FUNCTION_BLOCK T_PMLSubUnitInfoCollection EXTENDS T_NamedBase IMPLEMENTS I_PMLSubUnitInfo
VAR
	_info : ST_PMLSubUnitInfo;
	baseCollection : T_CollectionBase;
END_VAR

METHOD AddUnit : BOOL
VAR_INPUT
	newUnit : I_PMLSubUnitInfo;
END_VAR
IF newUnit = 0 THEN
	LogError( 'Cannot AddUnit invalid ref' );
	RETURN;
END_IF

AddUnit := baseCollection.AddItem( newItem := CastToBase(newUnit) );
END_METHOD

METHOD PRIVATE CastToBase : I_InterfaceBase
VAR_INPUT
	Unit : I_PMLSubUnitInfo;
END_VAR
__QUERYINTERFACE(Unit, CastToBase);
END_METHOD

METHOD CastToType : I_PMLSubUnitInfo
VAR_INPUT
	Base : I_InterfaceBase;
END_VAR
__QUERYINTERFACE(Base, CastToType);
END_METHOD

METHOD TryGetUnit: BOOL
VAR_INPUT
	index : UDINT;
END_VAR
VAR_OUTPUT
	Unit : I_PMLSubUnitInfo;
END_VAR
VAR
	baseItem : I_InterfaceBase;
END_VAR
baseCollection.TryGetItem(index, item => baseItem);
Unit := CastToType(baseItem);

IF Unit = 0 THEN
	LogError( 'Cannot TryGetUnit  Unit = 0' );
	RETURN;
END_IF 

TryGetUnit := Unit <> 0;
END_METHOD

END_FUNCTION_BLOCK

(* stored: Version 1.1.0.1, ProductVersion 3.1.4024.12
   POU T_PMLSubUnitInfoCollection: Id {ccfaf873-a746-4d0e-80b9-d4c09c831a9a}, SpecialFunc None
   Folder Private: Id {b080cbbd-bebb-4f49-af56-eee791651d6e}
   Method AddUnit: Id {edbc1f8a-3500-4b7c-bdb7-60b253486aba}
   Method CastToBase: Id {30ce565b-3c82-4a28-94a9-23dcbd458f22}
   Method CastToType: Id {a31f73da-5b42-475a-a9a5-d1ed373431f1}
   Method TryGetUnit: Id {608b8c09-7058-4b13-8e8e-aa3c05cb56c3} *)
